(* CODESYS project TcDynCollections.library
   Company: FisoThemes
   DefaultNamespace: TcDynCollections
   Version: 0.2.0.0
   DocFormat: reStructuredText
   Placeholder: TwinCat Dynamic Collections
   Author: Goodwill Mzumala
   Description: A library for handling collections of data dynamically.
   Title: TwinCat Dynamic Collections

Project tree, tasks and I/O mapping:
  libraries: Tc2_Standard, * (Beckhoff Automation GmbH); Tc2_System, * (Beckhoff Automation GmbH); Tc3_Module, * (Beckhoff Automation GmbH); Tc2_Utilities, 3.3.38.0 (Beckhoff Automation GmbH)
  DUTs/
    Interfaces/
      interface I_Collections: _Count, _Error_Status, _Is_Empty, Clear
      interface I_List: Add_Back, Add_Front, Find, Get, Get_First, Get_Value_As_String, Insert, Remove, RemoveAt, Resize, Reverse, Set
      interface I_List_ReadOnly: _Count, _Is_Empty, Find, Get, Get_First, Get_Value_As_String
      interface I_List_WriteOnly: Add_Back, Add_Front, Clear, Insert, Remove, RemoveAt, Resize, Reverse, Set
      interface I_Queue: Dequeue, Dequeue_Void, Enqueue, Enqueue_At_Front, Peek, Reverse
      interface I_Stack: Peek, Pop, Pop_Void, Push, Reverse, Top
    Structs/
      data type ST_ERROR
      data type ST_GENERIC
      data type ST_NODE
  GVLs/
  POUs/
    Examples/
      program P_Array_List_Example [ST]
      program P_List_Example [ST]
      program P_Queue_Example [ST]
      program P_Stack_Example [ST]
    Function Blocks/
      function block FB_Array_List [ST]: ClearException, EmptyListException, LessThanZeroException, MemCmpErrExpection, OutOfBoundsException, TypeMismatchException, CopyValueTo, DecrementCount, Free_Value, GetValueAsString, IncrementCount, Malloc_Array, Malloc_Value, SetValue, _Is_Empty, Add_Back, Add_Front, Clear, FB_exit, FB_init, Find, Get, Get_First, Get_Value_As_String, Insert, Remove, RemoveAt, Resize, Reverse, Set
      function block FB_Collections [ST]: _Count, _Error_Status, _Is_Empty, Clear
      function block FB_List [ST]: ClearException, EmptyListException, MemCmpErrExpection, OutOfBoundsException, TypeMismatchException, CopyValueTo, DecrementCount, Free_Node, GetValueAsString, IncrementCount, Iterate, Malloc_Node, SetValue, _Is_Empty, Add_Back, Add_Front, Clear, FB_exit, FB_init, Find, Get, Get_First, Get_Value_As_String, Insert, Remove, RemoveAt, Resize, Reverse, Set
      function block FB_Queue [ST]: _Count, _Is_Empty, CatchError, Clear, Dequeue, Dequeue_Void, Enqueue, Enqueue_At_Front, Peek, Reverse
      function block FB_Stack [ST]: _Count, _Is_Empty, CatchError, Clear, Peek, Pop, Pop_Void, Push, Reverse, Top
    program MAIN [ST]
  Project Information/
    function F_GetCompany [ST]
    function F_GetTitle [ST]
    function F_GetVersion [ST]
  UML/
    Array List UML
    Collections UML
    List UML
    Queue UML
    Stack UML
  Version/
    global variables Global_Version
  VISUs/
*)

// DUTs/Structs/ST_ERROR
(* STRUCT used to contain error status information. *)
{attribute 'enable_dynamic_creation'}
TYPE ST_ERROR :
STRUCT
	bSTATUS : BOOL; 		// Indicates if an error has occurred | TRUE = error, FALSE = no error
	nCODE 	: DINT; 		// Error code specific to the particular error.
	sSOURCE : T_MaxString; 	// Textual information describing the error.
END_STRUCT
END_TYPE

// DUTs/Structs/ST_GENERIC
(* Generic data type used for Programs/Functions/Function Blocks to handle data in a generic way. *)
{attribute 'enable_dynamic_creation'}
TYPE ST_GENERIC EXTENDS __SYSTEM.AnyType :
STRUCT
	sValue : T_MaxString; 	// Data of parameter as a string for easy convertion.
END_STRUCT
END_TYPE

// DUTs/Structs/ST_NODE
(* Node for linked list*)
{attribute 'enable_dynamic_creation'}
TYPE ST_NODE:
STRUCT
	Data 	: ST_GENERIC; // Stored data.
	pNext 	: POINTER TO ST_NODE := Tc3_Module.GVL.NULL; 	// Pointer to next node.
END_STRUCT
END_TYPE

// Version/Global_Version
{attribute 'TcGenerated'}
{attribute 'no-analysis'}
{attribute 'linkalways'}
// This function has been automatically generated from the project information.
VAR_GLOBAL CONSTANT
	{attribute 'const_non_replaced'}
	stLibVersion_TwinCat_Dynamic_Collections : ST_LibVersion := (iMajor := 0, iMinor := 2, iBuild := 0, iRevision := 0, nFlags := 0, sVersion := '0.2.0.0');
END_VAR

// DUTs/Interfaces/I_Collections
INTERFACE I_Collections

// Number of items in the collection
PROPERTY _Count : DINT
GET
END_GET
END_PROPERTY

(* Gets collection's error status *)
PROPERTY _Error_Status : ST_ERROR
GET
END_GET
END_PROPERTY

// Checks if collection is empty
PROPERTY _Is_Empty : BOOL
GET
END_GET
END_PROPERTY

// Empties/Clears/Deletes every item in the collection
METHOD Clear
END_METHOD

END_INTERFACE

// DUTs/Interfaces/I_List
INTERFACE I_List EXTENDS I_Collections

// Adds an item to the end of the list
METHOD Add_Back : I_List
VAR_INPUT
	Item 	: ANY; // Item to store in list
END_VAR
END_METHOD

// Adds an item at the front of the list
METHOD Add_Front : I_List
VAR_INPUT
	Item 	: ANY; // Item to store in list
END_VAR
END_METHOD

// Find the location of an item in list.
METHOD Find : I_List
VAR_INPUT
	Item 	: ANY; // Item to find in list
END_VAR
VAR_OUTPUT
	nIndex	: DINT; //Location of item in list 
END_VAR
END_METHOD

// Gets item from list at specified location without removing it
METHOD Get : I_List
VAR_INPUT
	Return_Item 	: ANY;  // Variable to store returned item
	nIndex 			: DINT; // Location of item
END_VAR
END_METHOD

// Gets item at the front of the list 
METHOD Get_First : I_List
VAR_INPUT
	Return_Item 	: ANY; // Variable to store returned item
END_VAR
END_METHOD

// Returns item as a string, if type to string conversion is supported
METHOD Get_Value_As_String : I_List
VAR_INPUT
	nIndex	: DINT; // Location of item
END_VAR
VAR_OUTPUT
	sItem 	: T_MaxString; // Variable to store returned item
END_VAR
END_METHOD

// Adds new item to list at specified location, if index = 0, item will be added at the front, if index = count, item will be added at the back
METHOD Insert : I_List
VAR_INPUT
	Item 	: ANY;  // Item to store in list
	nIndex 	: DINT; // Location of item
END_VAR
END_METHOD

// Removes item at the front of the list and returns nothing
METHOD Remove : I_List
END_METHOD

// Remove item at specified location and return nothing
METHOD RemoveAt : I_List
VAR_INPUT
	nIndex : DINT; // Location of item
END_VAR
END_METHOD

// Manually resize list. If list becomes smaller, items on higher locations will be deleted.
METHOD Resize : I_List
VAR_INPUT
	nSize : DINT; // New size of list.
END_VAR
END_METHOD

// Reverses the order of items in the list
METHOD Reverse : I_List
END_METHOD

// Adds new item to list in the specified location without resizing list
METHOD Set : I_List
VAR_INPUT
	Item 	: ANY; 	// Item to store in list
	nIndex 	: DINT; // Location of item
END_VAR
END_METHOD

END_INTERFACE

// DUTs/Interfaces/I_List_ReadOnly
// Implement this with I_List to allow a list to be Read Only. 
INTERFACE I_List_ReadOnly

// Number of items in the collection
PROPERTY _Count : DINT
GET
END_GET
END_PROPERTY

// Checks if collection is empty
PROPERTY _Is_Empty : BOOL
GET
END_GET
END_PROPERTY

// Find the location of an item in list.
METHOD Find : I_List
VAR_INPUT
	Item 	: ANY; // Item to find in list
END_VAR
VAR_OUTPUT
	nIndex	: DINT; //Location of item in list 
END_VAR
END_METHOD

// Gets item from list at specified location without removing it
METHOD Get : I_List
VAR_INPUT
	Return_Item 	: ANY;  // Variable to store returned item
	nIndex 			: DINT; // Location of item
END_VAR
END_METHOD

// Gets item at the front of the list 
METHOD Get_First : I_List
VAR_INPUT
	Return_Item 	: ANY; // Variable to store returned item
END_VAR
END_METHOD

// Returns item as a string, if type to string conversion is supported
METHOD Get_Value_As_String : I_List
VAR_INPUT
	nIndex	: DINT; // Location of item
END_VAR
VAR_OUTPUT
	sItem 	: T_MaxString; // Variable to store returned item
END_VAR
END_METHOD

END_INTERFACE

// DUTs/Interfaces/I_List_WriteOnly
// Implement this with I_List to allow a list to be Write Only. 
INTERFACE I_List_WriteOnly

// Adds an item to the end of the list
METHOD Add_Back : I_List
VAR_INPUT
	Item 	: ANY; // Item to store in list
END_VAR
END_METHOD

// Adds an item at the front of the list
METHOD Add_Front : I_List
VAR_INPUT
	Item 	: ANY; // Item to store in list
END_VAR
END_METHOD

// Empties/Clears/Deletes every item in the collection
METHOD Clear
END_METHOD

// Adds new item to list at specified location, if index = 0, item will be added at the front, if index = count, item will be added at the back
METHOD Insert : I_List
VAR_INPUT
	Item 	: ANY;  // Item to store in list
	nIndex 	: DINT; // Location of item
END_VAR
END_METHOD

// Removes item at the front of the list and returns nothing
METHOD Remove : I_List
END_METHOD

// Remove item at specified location and return nothing
METHOD RemoveAt : I_List
VAR_INPUT
	nIndex : DINT; // Location of item
END_VAR
END_METHOD

// Manually resize list. If list becomes smaller, items on higher locations will be deleted.
METHOD Resize : I_List
VAR_INPUT
	nSize : DINT; // New size of list.
END_VAR
END_METHOD

// Reverses the order of items in the list
METHOD Reverse : I_List
END_METHOD

// Adds new item to list in the specified location without resizing list
METHOD Set : I_List
VAR_INPUT
	Item 	: ANY; 	// Item to store in list
	nIndex 	: DINT; // Location of item
END_VAR
END_METHOD

END_INTERFACE

// DUTs/Interfaces/I_Queue
INTERFACE I_Queue EXTENDS I_Collections

(* Gets and remove item at the front of the queue *)
METHOD Dequeue : I_Queue
VAR_INPUT
	Item : ANY; (* Variable to store returned item value *)
END_VAR
END_METHOD

(* Removes item at the front of the queue without returning anything *)
METHOD Dequeue_Void : I_Queue
VAR_INPUT
END_VAR
END_METHOD

(* Adds item at the back of the queue *)
METHOD Enqueue : I_Queue
VAR_INPUT
	Item : ANY; (* Variable containg data to store on the queue *)
END_VAR
END_METHOD

(* Adds item at the front of the queue *)
METHOD Enqueue_At_Front : I_Queue
VAR_INPUT
	Item : ANY; (* Variable containg data to store on the queue *)
END_VAR
END_METHOD

(* Get item from the queue without removing it. *)
METHOD Peek : I_Queue
VAR_INPUT
	Item 	: ANY; (* Variable to store returned item value *)
	nIndex 	: DINT; (* Location of item*)
END_VAR
END_METHOD

METHOD Reverse : I_Queue
VAR_INPUT
END_VAR
END_METHOD

END_INTERFACE

// DUTs/Interfaces/I_Stack
INTERFACE I_Stack EXTENDS I_Collections

(* Get item from stack without removing it. *)
METHOD Peek : I_Stack
VAR_INPUT
	Item 	: ANY; (* Variable to store returned item value *)
	nIndex 	: DINT; (* Location of item*)
END_VAR
END_METHOD

(* Gets and deletes item at the top of the stack *)
METHOD Pop : I_Stack
VAR_INPUT
	Item : ANY; (* Variable to store returned item value *)
END_VAR
END_METHOD

(* Removes item at the top of the stack without returning anything *)
METHOD Pop_Void : I_Stack
VAR_INPUT
END_VAR
END_METHOD

(* Add item to the top of the stack *)
METHOD Push : I_Stack
VAR_INPUT
	Item : ANY; (* Variable containg data to store on the stack *)
END_VAR
END_METHOD

(* Reverses order of items on stack *)
METHOD Reverse : I_Stack
VAR_INPUT
END_VAR
END_METHOD

(* Get item at the top of the stack without removing it. *)
METHOD Top : I_Stack
VAR_INPUT
	Item 	: ANY; (* Variable to store returned item value *)
END_VAR
END_METHOD

END_INTERFACE

// POUs/Examples/P_Array_List_Example
PROGRAM P_Array_List_Example
VAR
	eState 		: (IDLE, INSERT, REVERSE, RESIZE, GET, SET, FIND, CLEAR, ADD_FRONT, ADD_BACK, REMOVE, REMOVE_AT);
	fbArray_List: FB_Array_List(0);
	nFind 		: DINT;
	sData 		: WSTRING;
	sRTNData	: ARRAY[0..6] OF WSTRING;
	nCount 		: DINT;
	stError 	: ST_ERROR;
END_VAR

stError := fbArray_List._Error_Status;
CASE eState OF
	INSERT:
		sData := "Cats";	fbArray_List.Insert(sData, 0);
		sData := "Dogs";	fbArray_List.Insert(sData, 1);
		sData := "Ravens";	fbArray_List.Insert(sData, 2);
		sData := "Mollies";	fbArray_List.Insert(sData, 3);
	REVERSE:
		fbArray_List.Reverse();
	RESIZE:
		fbArray_List.Resize(3);
	GET: 
		fbArray_List
			.Get(sRTNData[0], 0)
			.Get(sRTNData[1], 1)
			.Get(sRTNData[2], 2)
			.Get(sRTNData[3], 3)
			.Get(sRTNData[4], 4)
			.Get(sRTNData[5], 5)
			.Get(sRTNData[6], 6);
	SET:
		sData := "Ravens";	fbArray_List.Set(sData, 0);
		sData := "Mollies";	fbArray_List.Set(sData, 1);
		sData := "Dogs";	fbArray_List.Set(sData, 2);
		sData := "Cats";	fbArray_List.Set(sData, 3);
	FIND:
		sData := "Dogs"; fbArray_List.Find(sData, nIndex => nFind);
	CLEAR:
		fbArray_List.Clear();
	ADD_FRONT:
		sData := "Pythons";fbArray_List.Add_Front(sData);
	ADD_BACK:
		sData := "Anacondas"; fbArray_List.Add_Back(sData);
	REMOVE:
		fbArray_List.Remove();
	REMOVE_AT:
		fbArray_List.RemoveAt(2);
END_CASE
nCount := fbArray_List._Count;
eState := IDLE;

END_PROGRAM

// POUs/Function Blocks/FB_Array_List
(* A dynamic array that holds data of multiple types and can grow or shrink at run time. *)
FUNCTION_BLOCK FB_Array_List EXTENDS FB_Collections IMPLEMENTS I_List, I_List_ReadOnly, I_List_WriteOnly
VAR
	pData 		: POINTER TO ST_GENERIC;
END_VAR
VAR CONSTANT
	{warning disable C0228}
	stData 		: ST_GENERIC := (TypeClass := __SYSTEM.TYPE_CLASS.TYPE_NONE);
END_VAR

METHOD PROTECTED ClearException : BOOL;
VAR
END_VAR
ClearException 	:= stError.bSTATUS := FALSE;
stError.nCODE 	:= 0;
stError.sSOURCE := 'No error.';
END_METHOD

// Raises an expection if list is empty
METHOD PROTECTED EmptyListException : BOOL
VAR_INPUT
END_VAR
IF THIS^._Is_Empty THEN
	stError.bSTATUS := TRUE;
	stError.nCODE 	:= 2936;
	stError.sSOURCE := 'List is empty';
ELSE
	This^.ClearException();
	END_IF
EmptyListException := stError.bSTATUS;
END_METHOD

METHOD PROTECTED LessThanZeroException : BOOL
VAR_INPUT
	nIndex : DINT;
END_VAR
IF (nIndex < 0) THEN
	stError.bSTATUS := TRUE;
	stError.nCODE 	:= 5365;
	stError.sSOURCE := 'Out of bounds. Index is less than zero.';
ELSE
	This^.ClearException();
	END_IF
LessThanZeroException := stError.bSTATUS;
END_METHOD

// Compares memory sizes of 2 addresses. Returns TRUE  and raises error flag if theyre not same size.
METHOD PROTECTED MemCmpErrExpection : BOOL
VAR_INPUT
	pDestAddr,
	pSrcAddr 	: PVOID;
	nSize 		: UDINT;
END_VAR
VAR_INST
	nMemErr : DINT;
END_VAR
nMemErr := MEMCMP(pDestAddr, pSrcAddr, nSize);
IF nMemErr = -1 THEN 
	stError.bSTATUS := TRUE;
	stError.nCODE 	:= 4129;
	stError.sSOURCE := 'Incorrect parameter values. Destination address smaller than source address';
	
ELSIF nMemErr = 0 THEN THIS^.ClearException();
	
ELSIF nMemErr = 1 THEN
	stError.bSTATUS := TRUE;
	stError.nCODE 	:= 4823;
	stError.sSOURCE := 'Incorrect parameter values. Destination address greater that source address';

ELSE
	stError.bSTATUS := TRUE;
	stError.nCODE 	:= 4564;
	stError.sSOURCE := 'Incorrect parameter values. Pointer to destination/source address is NULL or allocated address memory is NULL.';
	END_IF

MemCmpErrExpection := stError.bSTATUS;
END_METHOD

METHOD PROTECTED OutOfBoundsException : BOOL
VAR_INPUT
	nIndex : DINT;
END_VAR
IF (nIndex < 0) OR (nIndex >= THIS^._Count) THEN
	stError.bSTATUS := TRUE;
	stError.nCODE 	:= 5374;
	stError.sSOURCE := 'Out of bounds. You tried to access data outside the range of this list.';
ELSE
	This^.ClearException();
	END_IF
OutOfBoundsException := stError.bSTATUS;
END_METHOD

METHOD TypeMismatchException : BOOL
VAR_INPUT
	Dest,
	Src 	: __SYSTEM.AnyType;
END_VAR
IF Dest.diSize <> Src.diSize THEN
	stError.bSTATUS := TRUE;
	stError.nCODE 	:= 3172;
	stError.sSOURCE := 'Type mismatch. Byte sizes are not the same';
ELSIF Dest.TypeClass <> Src.TypeClass THEN
	stError.bSTATUS := TRUE;
	stError.nCODE 	:= 3172;
	stError.sSOURCE := 'Type mismatch. Type classes are not the same';
ELSE
	THIS^.ClearException();
END_IF
TypeMismatchException := stError.bSTATUS;
END_METHOD

// Copy data from source memory space to desination memory space
METHOD PROTECTED CopyValueTo
VAR_INPUT
	Dest, Src 	: __SYSTEM.AnyType;
END_VAR
MEMMOVE(Dest.pValue, Src.pValue, TO_UDINT(Src.diSize));
END_METHOD

// Decrement list size by 1.
METHOD PROTECTED DecrementCount
VAR_INPUT
END_VAR
THIS^.nCount := THIS^.nCount - 1;
END_METHOD

// Deletes/frees Generic value's value from memory
METHOD PROTECTED Free_Value
VAR_INPUT
	Variable : __SYSTEM.AnyType;
END_VAR
IF Variable.pValue = 0 THEN RETURN; END_IF
__DELETE(Variable.pValue);
END_METHOD

METHOD PROTECTED GetValueAsString : T_MaxString
VAR_INPUT
	 Value : __SYSTEM.AnyType;
END_VAR
VAR	
	pBool			: POINTER TO BOOL;
    pByte			: POINTER TO BYTE;
    pWord			: POINTER TO WORD;
    pDWord			: POINTER TO DWORD;
    pLWord			: POINTER TO LWORD;
    pSint			: POINTER TO SINT;
    pInt			: POINTER TO INT;
    pDint			: POINTER TO DINT;
    pLint			: POINTER TO LINT;
    pUSint			: POINTER TO USINT;
    pUInt			: POINTER TO UINT;
    pUDint			: POINTER TO UDINT;
    pULint			: POINTER TO ULINT;
    pReal			: POINTER TO REAL;
    pLReal			: POINTER TO LREAL;
    pString			: POINTER TO STRING(255);
    pWString		: POINTER TO WSTRING;
    pTime			: POINTER TO TIME;
    pDate			: POINTER TO DATE;
    pDate_And_Time	: POINTER TO DATE_AND_TIME;
    pTime_Of_Day	: POINTER TO TIME_OF_DAY;
    pPointer		: PVOID;
	pLTime 			: POINTER TO LTIME;
END_VAR
IF Value.pValue = 0 THEN GetValueAsString := 'NULL'; RETURN; END_IF;

CASE Value.TypeClass OF 
	__SYSTEM.TYPE_CLASS.TYPE_BOOL:
		pBool := Value.pValue;
		GetValueAsString := TO_STRING(pBool^);
		
    __SYSTEM.TYPE_CLASS.TYPE_BYTE:
		pByte := Value.pValue;
		GetValueAsString := TO_STRING(pByte^);
		
    __SYSTEM.TYPE_CLASS.TYPE_WORD:
		pWord := Value.pValue;
		GetValueAsString := TO_STRING(pWord^);
		
    __SYSTEM.TYPE_CLASS.TYPE_DWORD:
		pDWord := Value.pValue;
		GetValueAsString := TO_STRING(pDWord^);
		
    __SYSTEM.TYPE_CLASS.TYPE_LWORD:
		pLWord := Value.pValue;
		GetValueAsString := TO_STRING(pLWord^);
		
    __SYSTEM.TYPE_CLASS.TYPE_SINT:
		pSint := Value.pValue;
		GetValueAsString := TO_STRING(pSint^);
		
    __SYSTEM.TYPE_CLASS.TYPE_INT:
		pInt := Value.pValue;
		GetValueAsString := TO_STRING(pInt^);
		
    __SYSTEM.TYPE_CLASS.TYPE_DINT:
		pDint := Value.pValue;
		GetValueAsString := TO_STRING(pDint^);
		
    __SYSTEM.TYPE_CLASS.TYPE_LINT:
		pLint := Value.pValue;
		GetValueAsString := TO_STRING(pLint^);
		
    __SYSTEM.TYPE_CLASS.TYPE_USINT:
		pUSint := Value.pValue;
		GetValueAsString := TO_STRING(pUSint^);
		
    __SYSTEM.TYPE_CLASS.TYPE_UINT:
		pUInt := Value.pValue;
		GetValueAsString := TO_STRING(pUInt^);
		
    __SYSTEM.TYPE_CLASS.TYPE_UDINT:
		pUDint := Value.pValue;
		GetValueAsString := TO_STRING(pUDint^);
		
    __SYSTEM.TYPE_CLASS.TYPE_ULINT:
		pULint := Value.pValue;
		GetValueAsString := TO_STRING(pULint^);
		
   __SYSTEM.TYPE_CLASS.TYPE_REAL:
		pReal := Value.pValue;
		GetValueAsString := TO_STRING(pReal^);
		
    __SYSTEM.TYPE_CLASS.TYPE_LREAL:
		pLReal := Value.pValue;
		GetValueAsString := TO_STRING(pLReal^);
		
    __SYSTEM.TYPE_CLASS.TYPE_STRING:
		pString := Value.pValue;
		GetValueAsString := TO_STRING(pString^);
		
   __SYSTEM.TYPE_CLASS.TYPE_WSTRING:
		pWString := Value.pValue;
		GetValueAsString := TO_STRING(pWString^);
		
    __SYSTEM.TYPE_CLASS.TYPE_TIME:
		pTime := Value.pValue;
		GetValueAsString := TO_STRING(pTime^);
		
    __SYSTEM.TYPE_CLASS.TYPE_DATE:
		pDate := Value.pValue;
		GetValueAsString := TO_STRING(pDate^);
		
    __SYSTEM.TYPE_CLASS.TYPE_DATEANDTIME:
		pDate_And_Time := Value.pValue;
		GetValueAsString := TO_STRING(pDate_And_Time^);
		
    __SYSTEM.TYPE_CLASS.TYPE_TIMEOFDAY:
		pTime_Of_Day := Value.pValue;
		GetValueAsString := TO_STRING(pTime_Of_Day^);
	
	__SYSTEM.TYPE_CLASS.TYPE_POINTER:
		GetValueAsString := TO_STRING(Value.pValue);
		
	__SYSTEM.TYPE_CLASS.TYPE_LTIME:
		pLTime := Value.pValue;
		GetValueAsString := TO_STRING(pLTime^);
ELSE
	GetValueAsString := 'TYPE TO STRING CONVERSION NOT SUPPORTED BY THIS TYPE'; 
END_CASE
END_METHOD

// Increments list size by 1
METHOD PROTECTED IncrementCount
VAR_INPUT
END_VAR
THIS^.nCount := THIS^.nCount + 1;
END_METHOD

// Allocate memory space for Array of Generics on the heap, returns Pointer to start of Generic Array;
// WARNING!!! Always have a place to store the return otherwise a memory leak will occur.
METHOD PROTECTED Malloc_Array : POINTER TO ST_GENERIC
VAR_INPUT
	nSize : DINT; // Array Size
END_VAR
VAR
	i, nByte_Size: DINT;
END_VAR
VAR CONSTANT
	{warning disable C0228}
	stData 		: ST_GENERIC;
END_VAR
nByte_Size := SIZEOF(ST_GENERIC)*nSize;
Malloc_Array := __NEW(BYTE, TO_UDINT(nByte_Size));
END_METHOD

// Allocate memory space for the Generic value's data on the heap, returns Generic;
// WARNING!!! Always have a place to store the return otherwise a memory leak will occur.
METHOD PROTECTED Malloc_Value : ST_GENERIC
VAR_INPUT
	Variable : __SYSTEM.AnyType;
END_VAR
Malloc_Value.sValue 	:= THIS^.GetValueAsString(Variable);
Malloc_Value.pValue 	:= __NEW(BYTE, TO_UDINT(Variable.diSize)); // Allocate space in memory to store data value.
Malloc_Value.diSize 	:= Variable.diSize;
Malloc_Value.TypeClass 	:= Variable.TypeClass;
END_METHOD

(* Set value of __SYSTEM.Anytype variable *)
METHOD PROTECTED SetValue
VAR_INPUT
	Variable	: __SYSTEM.Anytype;
	Value 		: USINT; // Character/byte to set.
END_VAR
MEMSET(Variable.pValue, Value, TO_UDINT(Variable.diSize));
END_METHOD

(* Checks of list is empty.*)
PROPERTY _Is_Empty : BOOL
GET
_Is_Empty := THIS^.nCount = 0;
END_GET
END_PROPERTY

// Adds an item to the end of the list
METHOD Add_Back : I_List
VAR_INPUT
	Item 	: ANY; // Item to store in list
END_VAR
Add_Back := THIS^;
IF THIS^._Is_Empty THEN THIS^.FB_init(FALSE,FALSE, 1); THIS^.Set(Item, 0); RETURN; END_IF
THIS^.Resize(THIS^._Count+1);
THIS^.Free_Value(THIS^.pData[THIS^._Count-1]);
THIS^.pData[THIS^._Count-1] := THIS^.Malloc_Value(Item);
THIS^.CopyValueTo(THIS^.pData[THIS^._Count-1], Item);
END_METHOD

// Adds an item at the front of the list
METHOD Add_Front : I_List
VAR_INPUT
	Item 	: ANY; // Item to store in list
END_VAR
VAR
	pOld_Data : POINTER TO ST_GENERIC;
	i : DINT;
END_VAR
Add_Front := THIS^;
IF THIS^._Is_Empty THEN THIS^.FB_init(FALSE,FALSE, 1); THIS^.Set(Item, 0); RETURN; END_IF

pOld_Data := THIS^.pData;
THIS^.pData := THIS^.Malloc_Array(THIS^._Count+1);

FOR i := 1 TO THIS^._Count DO
	THIS^.pData[i] := THIS^.Malloc_Value(pOld_Data[i-1]);
	THIS^.CopyValueTo(THIS^.pData[i], pOld_Data[i-1]);
	THIS^.Free_Value(pOld_Data[i-1]);
	END_FOR
__DELETE(pOld_Data);
THIS^.Set(Item, 0);
THIS^.IncrementCount();
END_METHOD

// Empties/Clears/Deletes every item in the list
METHOD Clear
VAR
	i : DINT;
END_VAR
IF NOT(THIS^._Is_Empty) THEN 
	FOR i := 0 TO THIS^._Count - 1 DO THIS^.Free_Value(THIS^.pData[i]); END_FOR
	__DELETE(THIS^.pData); 
	THIS^.nCount := 0; 
	END_IF
END_METHOD

METHOD FB_exit : BOOL
VAR_INPUT
	bInCopyCode : BOOL; // if TRUE, the exit method is called for exiting an instance that is copied afterwards (online change).
END_VAR
THIS^.Clear();
END_METHOD

METHOD FB_init : BOOL
VAR_INPUT
	bInitRetains 	: BOOL; // if TRUE, the retain variables are initialized (warm start / cold start)
	bInCopyCode 	: BOOL; // if TRUE, the instance afterwards gets moved into the copy code (online change)
	nLength 		: DINT; // Length to initialise array with.
END_VAR
VAR
	i, nByte_Size 	: DINT;
END_VAR
THIS^.Clear();
IF nLength <= 0 THEN RETURN; END_IF
THIS^.nCount := nLength;
THIS^.pData := THIS^.Malloc_Array(nLength);
END_METHOD

// Find the location of an item in list.
METHOD Find : I_List
VAR_INPUT
	Item 	: ANY; // Item to find in list
END_VAR
VAR_OUTPUT
	nIndex	: DINT; //Location of item in list 
END_VAR
VAR
	i : DINT;
	n : DINT := -1;
END_VAR
Find := THIS^;
IF THIS^.EmptyListException() THEN nIndex := -1; RETURN; END_IF
FOR i := 0 TO THIS^._Count-1 DO
	IF (THIS^.pData[i].pValue = 0) 					 THEN CONTINUE; END_IF
	IF (Item.TypeClass <> THIS^.pData[i].TypeClass) THEN CONTINUE; END_IF
	IF (Item.pValue^ <> THIS^.pData[i].pValue^) 	 THEN CONTINUE; END_IF
	
	CASE Item.TypeClass OF
		__SYSTEM.TYPE_CLASS.TYPE_STRING:
			IF LEN2(Item.pValue) <> LEN2(THIS^.pData[i].pValue) THEN CONTINUE; END_IF
			n := MEMCMP(Item.pValue, THIS^.pData[i].pValue, LEN2(THIS^.pData[i].pValue)+1);
				
		__SYSTEM.TYPE_CLASS.TYPE_WSTRING:
			IF WLEN2(Item.pValue) <> WLEN2(THIS^.pData[i].pValue) THEN CONTINUE; END_IF
			n := MEMCMP(Item.pValue, THIS^.pData[i].pValue, (WLEN2(THIS^.pData[i].pValue)*SIZEOF(WORD))+1);
	ELSE
		IF (Item.diSize <> THIS^.pData[i].diSize) THEN CONTINUE; END_IF	
		n := MEMCMP(Item.pValue, THIS^.pData[i].pValue, TO_UDINT(Item.diSize));
		END_CASE
		IF n = 0 THEN nIndex := i; RETURN; END_IF
	END_FOR
nIndex := -1;
END_METHOD

// Gets item at specified location;
METHOD Get : I_List
VAR_INPUT
	Return_Item 	: ANY;  // Variable to store requested node value
	nIndex 			: DINT; // Location of node
END_VAR
VAR_INST
	data : ST_GENERIC;
END_VAR
Get := THIS^;
IF THIS^.EmptyListException() OR THIS^.OutOfBoundsException(nIndex) THEN THIS^.SetValue(Return_Item, 16#0); RETURN; END_IF
IF THIS^.TypeMismatchException(Return_Item, THIS^.pData[nIndex]) THEN THIS^.SetValue(Return_Item, 16#0); RETURN; END_IF
THIS^.CopyValueTo(Return_Item, THIS^.pData[nIndex]);
END_METHOD

// Gets item at the front of the list 
METHOD Get_First : I_List
VAR_INPUT
	Return_Item 	: ANY; // Variable to store returned item
END_VAR
Get_First := THIS^;
THIS^.Get(Return_Item, 0);
END_METHOD

// Returns item as a string, if type to string conversion is supported
METHOD Get_Value_As_String : I_List
VAR_INPUT
	nIndex	: DINT; // Location of item
END_VAR
VAR_OUTPUT
	sItem 	: T_MaxString; // Variable to store returned item
END_VAR
Get_Value_As_String := THIS^;
IF THIS^.EmptyListException() OR THIS^.OutOfBoundsException(nIndex) THEN sItem := 'ERR: List is Empty or index Out of Bounds'; RETURN; END_IF
sItem := THIS^.pData[nIndex].sValue;
END_METHOD

// Adds new item to list at specified location, if index = 0, item will be added at the front, if index = count, item will be added at the back
METHOD Insert : I_List
VAR_INPUT
	Item 	: ANY;  // Item to store in list
	nIndex 	: DINT; // Location of item
END_VAR
VAR
	pOld_Data : POINTER TO ST_GENERIC;
	i : DINT;
END_VAR
Insert := THIS^;
IF nIndex = 0 THEN THIS^.Add_Front(Item); RETURN; END_IF
IF nIndex = THIS^._Count THEN THIS^.Add_Back(Item); RETURN; END_IF
IF THIS^.OutOfBoundsException(nIndex) THEN RETURN; END_IF

pOld_Data := THIS^.pData;
THIS^.pData := THIS^.Malloc_Array(THIS^._Count+1);
THIS^.IncrementCount();

FOR i := 0 TO nIndex-1 DO
	THIS^.pData[i] := THIS^.Malloc_Value(pOld_Data[i]);
	THIS^.CopyValueTo(THIS^.pData[i], pOld_Data[i]);
	THIS^.Free_Value(pOld_Data[i]);
	END_FOR
	
THIS^.Set(Item, nIndex);
	
FOR i := nIndex+1 TO THIS^._Count-1 DO
	THIS^.pData[i] := THIS^.Malloc_Value(pOld_Data[i-1]);
	THIS^.CopyValueTo(THIS^.pData[i], pOld_Data[i-1]);
	THIS^.Free_Value(pOld_Data[i-1]);
	END_FOR
__DELETE(pOld_Data);
END_METHOD

// Removes item at the front of the list and returns nothing
METHOD Remove : I_List
VAR
	i : DINT;
END_VAR
Remove := THIS^;
IF THIS^.EmptyListException() THEN RETURN; END_IF
IF THIS^._Count = 1 THEN THIS^.Clear(); RETURN; END_IF;
THIS^.Free_Value(THIS^.pData[0]);
FOR i := 0 TO THIS^._Count-2 DO THIS^.pData[i] := THIS^.pData[i+1]; END_FOR
THIS^.Resize(THIS^._Count-1);
END_METHOD

// Remove item at specified location and return nothing
METHOD RemoveAt : I_List
VAR_INPUT
	nIndex : DINT; // Location of item
END_VAR
VAR
	i : DINT;
END_VAR
RemoveAt := THIS^;
IF THIS^.EmptyListException() THEN RETURN; END_IF
IF THIS^.OutOfBoundsException(nIndex) THEN RETURN; END_IF
IF nIndex = 0 THEN THIS^.Remove(); RETURN; END_IF
IF nIndex = THIS^._Count - 1 THEN THIS^.Resize(THIS^._Count - 1); RETURN; END_IF
THIS^.Free_Value(THIS^.pData[nIndex]);
FOR i := nIndex TO THIS^._Count-1 DO THIS^.pData[i] := THIS^.pData[i+1]; END_FOR
THIS^.Resize(THIS^._Count-1);
END_METHOD

// Manually resize list. If list becomes smaller, items on higher locations will be deleted.
METHOD Resize : I_List
VAR_INPUT
	nSize : DINT; // New size of list.
END_VAR
VAR
	pOld_Data 		: POINTER TO ST_GENERIC;
	i,
	nOld_Data_Count, 
	nByte_Size : DINT;
END_VAR
Resize := THIS^;
IF THIS^.LessThanZeroException(nSize) THEN RETURN; END_IF
IF (nSize = 0) THEN THIS^.Clear(); RETURN; END_IF
IF nSize = THIS^._Count THEN RETURN; END_IF
IF THIS^._Is_Empty THEN THIS^.FB_init(FALSE,FALSE, nSize); RETURN; END_IF

pOld_Data 		:= THIS^.pData;
nOld_Data_Count := THIS^._Count;

THIS^.pData := THIS^.Malloc_Array(nSize);

FOR i := 0 TO nSize - 1 DO
	IF (i = nOld_Data_Count) AND (nSize > nOld_Data_Count) THEN EXIT; END_IF
	THIS^.pData[i] := THIS^.Malloc_Value(pOld_Data[i]);
	THIS^.CopyValueTo(THIS^.pData[i], pOld_Data[i]);
	THIS^.Free_Value(pOld_Data[i]);
	END_FOR
__DELETE(pOld_Data);
THIS^.nCount := nSize;
END_METHOD

// Reverses the order of items in the list
METHOD Reverse : I_List
VAR
	pOld_Data 	: POINTER TO ST_GENERIC;
	nByte_Size 	: DINT;
	i			: DINT;
END_VAR
Reverse := THIS^;
IF THIS^.EmptyListException() THEN RETURN; END_IF
IF THIS^._Count = 1 THEN RETURN; END_IF

pOld_Data 	:= THIS^.pData;

THIS^.pData := THIS^.Malloc_Array(THIS^._Count);

FOR i:= 0 TO THIS^._Count - 1 DO
	THIS^.pData[i] := THIS^.Malloc_Value(pOld_Data[(THIS^._Count-1)-i]);
	THIS^.CopyValueTo(THIS^.pData[i], pOld_Data[(THIS^._Count-1)-i]);
	THIS^.Free_Value(pOld_Data[(THIS^._Count-1)-i]);
	END_FOR
__DELETE(pOld_Data);
END_METHOD

// Adds new item to list in the specified location without resizing list
METHOD Set : I_List
VAR_INPUT
	Item 	: ANY; 	// Item to store in list
	nIndex 	: DINT; // Location of item
END_VAR
Set := THIS^;
IF THIS^.OutOfBoundsException(nIndex) OR THIS^.EmptyListException() THEN RETURN; END_IF
THIS^.Free_Value(THIS^.pData[nIndex]);
THIS^.pData[nIndex] := THIS^.Malloc_Value(Item);
THIS^.CopyValueTo(THIS^.pData[nIndex], Item);
END_METHOD

END_FUNCTION_BLOCK

// POUs/Function Blocks/FB_Collections
FUNCTION_BLOCK ABSTRACT FB_Collections IMPLEMENTS I_Collections
VAR
	stError : ST_ERROR;
	nCount 	: DINT; // Size of Collection
END_VAR

(* Number of items in the collection *)
PROPERTY _Count : DINT
GET
_Count := THIS^.nCount;
END_GET
END_PROPERTY

(* Gets collection's error status *)
PROPERTY _Error_Status : ST_ERROR
GET
_Error_Status := THIS^.stError;
END_GET
END_PROPERTY

(* Checks if collection is empty.*)
PROPERTY _Is_Empty : BOOL
GET
END_GET
END_PROPERTY

(* Empties/Clears/Deletes every element on the collection*)
METHOD Clear
END_METHOD

END_FUNCTION_BLOCK

// POUs/Examples/P_List_Example
PROGRAM P_List_Example
VAR
	eState 		: (IDLE, INSERT, REVERSE, RESIZE, GET, SET, FIND, CLEAR, ADD_FRONT, ADD_BACK, REMOVE, REMOVE_AT);
	fbList 		: FB_List;
	nFind 		: DINT;
	sData 		: WSTRING;
	sRTNData	: ARRAY[0..6] OF WSTRING;
	nCount 		: DINT;
	stError 	: ST_ERROR;
END_VAR

stError := fbList._Error_Status;
CASE eState OF
	INSERT:
		sData := "Cats";	fbList.Insert(sData, 0);
		sData := "Dogs";	fbList.Insert(sData, 1);
		sData := "Ravens";	fbList.Insert(sData, 2);
		sData := "Mollies";	fbList.Insert(sData, 3);
	REVERSE:
		fbList.Reverse();
	RESIZE:
		fbList.Resize(3);
	GET: 
		fbList
			.Get(sRTNData[0], 0)
			.Get(sRTNData[1], 1)
			.Get(sRTNData[2], 2)
			.Get(sRTNData[3], 3)
			.Get(sRTNData[4], 4)
			.Get(sRTNData[5], 5)
			.Get(sRTNData[6], 6);
	SET:
		sData := "Ravens";	fbList.Set(sData, 0);
		sData := "Mollies";	fbList.Set(sData, 1);
		sData := "Dogs";	fbList.Set(sData, 2);
		sData := "Cats";	fbList.Set(sData, 3);
	FIND:
		sData := "Dogs"; fbList.Find(sData, nIndex => nFind);
	CLEAR:
		fbList.Clear();
	ADD_FRONT:
		sData := "Pythons";fbList.Add_Front(sData);
	ADD_BACK:
		sData := "Anacondas"; fbList.Add_Back(sData);
	REMOVE:
		fbList.Remove();
	REMOVE_AT:
		fbList.RemoveAt(2);
END_CASE
nCount := fbList._Count;
eState := IDLE;

END_PROGRAM

// POUs/Function Blocks/FB_List
// Dyanamic List that can store a collection of any types. Similiar to python lists.
FUNCTION_BLOCK FB_List EXTENDS FB_Collections IMPLEMENTS I_List, I_List_ReadOnly, I_List_WriteOnly
VAR
	pHead	: POINTER TO ST_NODE;
END_VAR

METHOD PROTECTED ClearException : BOOL;
VAR
END_VAR
ClearException 	:= stError.bSTATUS := FALSE;
stError.nCODE 	:= 0;
stError.sSOURCE := 'No error.';
END_METHOD

// Raises an expection if list is empty
METHOD PROTECTED EmptyListException : BOOL
VAR_INPUT
END_VAR
IF THIS^._Is_Empty THEN
	stError.bSTATUS := TRUE;
	stError.nCODE 	:= 2936;
	stError.sSOURCE := 'List is empty';
ELSE
	This^.ClearException();
	END_IF
EmptyListException := stError.bSTATUS;
END_METHOD

// Compares memory sizes of 2 addresses. Returns TRUE  and raises error flag if theyre not same size.
METHOD PROTECTED MemCmpErrExpection : BOOL
VAR_INPUT
	pDestAddr,
	pSrcAddr 	: PVOID;
	nSize 		: UDINT;
END_VAR
VAR_INST
	nMemErr : DINT;
END_VAR
nMemErr := MEMCMP(pDestAddr, pSrcAddr, nSize);
IF nMemErr = -1 THEN 
	stError.bSTATUS := TRUE;
	stError.nCODE 	:= 4129;
	stError.sSOURCE := 'Incorrect parameter values. Destination address smaller than source address';
	
ELSIF nMemErr = 0 THEN THIS^.ClearException();
	
ELSIF nMemErr = 1 THEN
	stError.bSTATUS := TRUE;
	stError.nCODE 	:= 4823;
	stError.sSOURCE := 'Incorrect parameter values. Destination address greater that source address';

ELSE
	stError.bSTATUS := TRUE;
	stError.nCODE 	:= 4564;
	stError.sSOURCE := 'Incorrect parameter values. Pointer to destination/source address is NULL or allocated address memory is NULL.';
	END_IF

MemCmpErrExpection := stError.bSTATUS;
END_METHOD

METHOD PROTECTED OutOfBoundsException : BOOL
VAR_INPUT
	nIndex : DINT;
END_VAR
IF (nIndex < 0) OR (nIndex >= THIS^._Count) THEN
	stError.bSTATUS := TRUE;
	stError.nCODE 	:= 5374;
	stError.sSOURCE := 'Out of bounds. You tried to access data outside the range of this list.';
ELSE
	This^.ClearException();
	END_IF
OutOfBoundsException := stError.bSTATUS;
END_METHOD

METHOD TypeMismatchException : BOOL
VAR_INPUT
	Dest,
	Src 	: __SYSTEM.AnyType;
END_VAR
IF Dest.diSize <> Src.diSize THEN
	stError.bSTATUS := TRUE;
	stError.nCODE 	:= 3172;
	stError.sSOURCE := 'Type mismatch. Byte sizes are not the same';
ELSIF Dest.TypeClass <> Src.TypeClass THEN
	stError.bSTATUS := TRUE;
	stError.nCODE 	:= 3172;
	stError.sSOURCE := 'Type mismatch. Type classes are not the same';
ELSE
	THIS^.ClearException();
END_IF
TypeMismatchException := stError.bSTATUS;
END_METHOD

// Copy data from source memory space to desination memory space
METHOD PROTECTED CopyValueTo
VAR_INPUT
	Dest, Src : __SYSTEM.AnyType;
END_VAR
MEMMOVE(Dest.pValue, Src.pValue, TO_UDINT(Dest.diSize));
END_METHOD

// Decrement list size by 1.
METHOD PROTECTED DecrementCount
VAR_INPUT
END_VAR
THIS^.nCount := THIS^.nCount - 1;
END_METHOD

// Deletes/frees node and it's value from memory
METHOD PROTECTED Free_Node
VAR_INPUT
	pNode : POINTER TO ST_NODE; 
END_VAR
__DELETE(pNode^.Data.pValue);
__DELETE(pNode);
END_METHOD

METHOD PROTECTED GetValueAsString : T_MaxString
VAR_INPUT
	 Value : __SYSTEM.AnyType;
END_VAR
VAR	
	pBool			: POINTER TO BOOL;
    pByte			: POINTER TO BYTE;
    pWord			: POINTER TO WORD;
    pDWord			: POINTER TO DWORD;
    pLWord			: POINTER TO LWORD;
    pSint			: POINTER TO SINT;
    pInt			: POINTER TO INT;
    pDint			: POINTER TO DINT;
    pLint			: POINTER TO LINT;
    pUSint			: POINTER TO USINT;
    pUInt			: POINTER TO UINT;
    pUDint			: POINTER TO UDINT;
    pULint			: POINTER TO ULINT;
    pReal			: POINTER TO REAL;
    pLReal			: POINTER TO LREAL;
    pString			: POINTER TO STRING(255);
    pWString		: POINTER TO WSTRING;
    pTime			: POINTER TO TIME;
    pDate			: POINTER TO DATE;
    pDate_And_Time	: POINTER TO DATE_AND_TIME;
    pTime_Of_Day	: POINTER TO TIME_OF_DAY;
    pPointer		: PVOID;
	pLTime 			: POINTER TO LTIME;
END_VAR
IF Value.pValue = 0 THEN GetValueAsString := 'NULL'; RETURN; END_IF;

CASE Value.TypeClass OF 
	__SYSTEM.TYPE_CLASS.TYPE_BOOL:
		pBool := Value.pValue;
		GetValueAsString := TO_STRING(pBool^);
		
    __SYSTEM.TYPE_CLASS.TYPE_BYTE:
		pByte := Value.pValue;
		GetValueAsString := TO_STRING(pByte^);
		
    __SYSTEM.TYPE_CLASS.TYPE_WORD:
		pWord := Value.pValue;
		GetValueAsString := TO_STRING(pWord^);
		
    __SYSTEM.TYPE_CLASS.TYPE_DWORD:
		pDWord := Value.pValue;
		GetValueAsString := TO_STRING(pDWord^);
		
    __SYSTEM.TYPE_CLASS.TYPE_LWORD:
		pLWord := Value.pValue;
		GetValueAsString := TO_STRING(pLWord^);
		
    __SYSTEM.TYPE_CLASS.TYPE_SINT:
		pSint := Value.pValue;
		GetValueAsString := TO_STRING(pSint^);
		
    __SYSTEM.TYPE_CLASS.TYPE_INT:
		pInt := Value.pValue;
		GetValueAsString := TO_STRING(pInt^);
		
    __SYSTEM.TYPE_CLASS.TYPE_DINT:
		pDint := Value.pValue;
		GetValueAsString := TO_STRING(pDint^);
		
    __SYSTEM.TYPE_CLASS.TYPE_LINT:
		pLint := Value.pValue;
		GetValueAsString := TO_STRING(pLint^);
		
    __SYSTEM.TYPE_CLASS.TYPE_USINT:
		pUSint := Value.pValue;
		GetValueAsString := TO_STRING(pUSint^);
		
    __SYSTEM.TYPE_CLASS.TYPE_UINT:
		pUInt := Value.pValue;
		GetValueAsString := TO_STRING(pUInt^);
		
    __SYSTEM.TYPE_CLASS.TYPE_UDINT:
		pUDint := Value.pValue;
		GetValueAsString := TO_STRING(pUDint^);
		
    __SYSTEM.TYPE_CLASS.TYPE_ULINT:
		pULint := Value.pValue;
		GetValueAsString := TO_STRING(pULint^);
		
   __SYSTEM.TYPE_CLASS.TYPE_REAL:
		pReal := Value.pValue;
		GetValueAsString := TO_STRING(pReal^);
		
    __SYSTEM.TYPE_CLASS.TYPE_LREAL:
		pLReal := Value.pValue;
		GetValueAsString := TO_STRING(pLReal^);
		
    __SYSTEM.TYPE_CLASS.TYPE_STRING:
		pString := Value.pValue;
		GetValueAsString := TO_STRING(pString^);
		
   __SYSTEM.TYPE_CLASS.TYPE_WSTRING:
		pWString := Value.pValue;
		GetValueAsString := TO_STRING(pWString^);
		
    __SYSTEM.TYPE_CLASS.TYPE_TIME:
		pTime := Value.pValue;
		GetValueAsString := TO_STRING(pTime^);
		
    __SYSTEM.TYPE_CLASS.TYPE_DATE:
		pDate := Value.pValue;
		GetValueAsString := TO_STRING(pDate^);
		
    __SYSTEM.TYPE_CLASS.TYPE_DATEANDTIME:
		pDate_And_Time := Value.pValue;
		GetValueAsString := TO_STRING(pDate_And_Time^);
		
    __SYSTEM.TYPE_CLASS.TYPE_TIMEOFDAY:
		pTime_Of_Day := Value.pValue;
		GetValueAsString := TO_STRING(pTime_Of_Day^);
	
	__SYSTEM.TYPE_CLASS.TYPE_POINTER:
		GetValueAsString := TO_STRING(Value.pValue);
		
	__SYSTEM.TYPE_CLASS.TYPE_LTIME:
		pLTime := Value.pValue;
		GetValueAsString := TO_STRING(pLTime^);
ELSE
	GetValueAsString := 'TYPE TO STRING CONVERSION NOT SUPPORTED BY THIS TYPE'; 
END_CASE
END_METHOD

// Increments list size by 1
METHOD PROTECTED IncrementCount
VAR_INPUT
END_VAR
THIS^.nCount := THIS^.nCount + 1;
END_METHOD

// Returns pointer to node at specificied location;
METHOD PROTECTED Iterate : POINTER TO ST_NODE
VAR_INPUT
	nIndex : DINT;
END_VAR
VAR 
	i 		: DINT;
	pTemp 	: POINTER TO ST_NODE;
END_VAR
IF THIS^.OutOfBoundsException(nIndex) THEN RETURN; END_IF
IF nIndex = 0 THEN Iterate := THIS^.pHead; RETURN; END_IF
//IF nIndex = THIS^._Count-1 THEN Iterate := pTail; RETURN; END_IF
pTemp := pHead;
FOR i := 1 TO nIndex DO pTemp := pTemp^.pNext; END_FOR
Iterate := pTemp;
END_METHOD

// Allocate memory space for node and the value for it's data on the heap, returns pointer to node;
// WARNING!!! Always have a place to store the node pointer otherwise a memory leak will occur.
METHOD PROTECTED Malloc_Node : POINTER TO ST_NODE
VAR_INPUT
	Variable : __SYSTEM.AnyType;
END_VAR
VAR
	pTemp 	: POINTER TO ST_NODE;
END_VAR
pTemp 					:= __NEW(ST_NODE); // Allocate space in memory for a node.
pTemp^.Data.sValue 		:= THIS^.GetValueAsString(Variable);
pTemp^.Data.pValue 		:= __NEW(BYTE, TO_UDINT(Variable.diSize)); // Allocate space in memory to store data value.
pTemp^.Data.diSize 		:= Variable.diSize;
pTemp^.Data.TypeClass 	:= Variable.TypeClass;

Malloc_Node := pTemp;
END_METHOD

(* Set value of __SYSTEM.Anytype variable *)
METHOD PROTECTED SetValue
VAR_INPUT
	Variable	: __SYSTEM.Anytype;
	Value 		: USINT; // Character/byte to set.
END_VAR
MEMSET(Variable.pValue, Value, TO_UDINT(Variable.diSize));
END_METHOD

(* Checks of list is empty.*)
PROPERTY _Is_Empty : BOOL
GET
_Is_Empty := (THIS^._Count = 0) AND (THIS^.pHead = 0);
END_GET
END_PROPERTY

// Adds an item to the end of the list
METHOD Add_Back : I_List
VAR_INPUT
	Item 	: ANY; // Value to store in list
END_VAR
VAR
	pTemp 	: POINTER TO ST_NODE;
END_VAR
Add_Back := THIS^;
pTemp := THIS^.Malloc_Node(Item);
THIS^.CopyValueTo(pTemp^.Data, Item);

IF THIS^._Is_Empty THEN THIS^.pHead := pTemp;
ELSE Iterate(THIS^._Count - 1)^.pNext := pTemp; END_IF

THIS^.IncrementCount();
END_METHOD

// Adds an item at the front of the list
METHOD Add_Front : I_List
VAR_INPUT
	Item 	: ANY; // Item to store in list
END_VAR
VAR
	pTemp 	: POINTER TO ST_NODE;
END_VAR
Add_Front := THIS^;
pTemp := THIS^.Malloc_Node(Item);
THIS^.CopyValueTo(pTemp^.Data, Item);

pTemp^.pNext := THIS^.pHead; THIS^.pHead := pTemp;
THIS^.IncrementCount();
END_METHOD

(* Empties/Clears/Deletes every item in the list *)
METHOD Clear
VAR
	pTemp : POINTER TO ST_NODE;
END_VAR
pTemp := THIS^.pHead;
WHILE pTemp <> 0 DO
	pTemp := pTemp^.pNext; THIS^.Remove();
END_WHILE
END_METHOD

METHOD FB_exit : BOOL
VAR_INPUT
	(* if TRUE, the exit method is called for exiting an instance that is copied afterwards (online change).*)
	bInCopyCode	: BOOL;
END_VAR
This^.Clear();
END_METHOD

METHOD FB_init : BOOL
VAR_INPUT
	bInitRetains : BOOL; // if TRUE, the retain variables are initialized (warm start / cold start)
	bInCopyCode : BOOL;  // if TRUE, the instance afterwards gets moved into the copy code (online change)
END_VAR
THIS^.Clear();
THIS^.pHead := Tc3_Module.GVL.NULL;
END_METHOD

// Find the location of an item in list.
METHOD Find : I_List
VAR_INPUT
	Item 	: ANY; // Item to find in list
END_VAR
VAR_OUTPUT
	nIndex	: DINT; //Location of item in list 
END_VAR
VAR
	pTemp 	: POINTER TO ST_NODE;
	i 		: DINT;
	n 		: DINT := -1;
END_VAR
Find := THIS^;
IF THIS^.EmptyListException() THEN nIndex := -1; RETURN; END_IF
pTemp := THIS^.pHead;
FOR i := 0 TO THIS^._Count-1 DO
	IF pTemp = 0 THEN EXIT; END_IF
	IF (pTemp^.Data.pValue = 0) 					THEN pTemp := pTemp^.pNext; CONTINUE; END_IF
	IF (Item.TypeClass <> pTemp^.Data.TypeClass) 	THEN pTemp := pTemp^.pNext; CONTINUE; END_IF
	IF (Item.pValue^ <> pTemp^.Data.pValue^) 		THEN pTemp := pTemp^.pNext; CONTINUE; END_IF
	
	CASE Item.TypeClass OF
		__SYSTEM.TYPE_CLASS.TYPE_STRING:
			IF LEN2(Item.pValue) <> LEN2(pTemp^.Data.pValue) THEN pTemp := pTemp^.pNext; CONTINUE; END_IF
			n := MEMCMP(Item.pValue, pTemp^.Data.pValue, LEN2(pTemp^.Data.pValue)+1);
				
		__SYSTEM.TYPE_CLASS.TYPE_WSTRING:
			IF WLEN2(Item.pValue) <> WLEN2(pTemp^.Data.pValue) THEN pTemp := pTemp^.pNext; CONTINUE; END_IF
			n := MEMCMP(Item.pValue, pTemp^.Data.pValue, (WLEN2(pTemp^.Data.pValue)*SIZEOF(WORD))+1);
	ELSE
		IF (Item.diSize <> pTemp^.Data.diSize) THEN pTemp := pTemp^.pNext; CONTINUE; END_IF	
		n := MEMCMP(Item.pValue, pTemp^.Data.pValue, TO_UDINT(Item.diSize));
	END_CASE
	IF n = 0 THEN nIndex := i; RETURN; END_IF
	pTemp := pTemp^.pNext;
	END_FOR
nIndex := -1;
END_METHOD

// Gets item from list at specified location without removing it
METHOD Get : I_List
VAR_INPUT
	Return_Item 	: ANY;  // Variable to store returned item
	nIndex 			: DINT; // Location of item
END_VAR
VAR
	pTemp : POINTER TO ST_NODE;
END_VAR
Get := THIS^;
IF THIS^.EmptyListException() OR THIS^.OutOfBoundsException(nIndex) THEN THIS^.SetValue(Return_Item, 16#0); RETURN; END_IF
pTemp := Iterate(nIndex);
IF THIS^.TypeMismatchException(Return_Item, pTemp^.Data) THEN THIS^.SetValue(Return_Item, 16#0); RETURN; END_IF
THIS^.CopyValueTo(Return_Item, pTemp^.Data);
END_METHOD

// Gets item at the front of the list 
METHOD Get_First : I_List
VAR_INPUT
	Return_Item 	: ANY; // Variable to store returned item
END_VAR
VAR
	pTemp 	: POINTER TO ST_NODE;
END_VAR
Get_First := THIS^;
IF THIS^.TypeMismatchException(Return_Item, pHead^.Data) OR THIS^.EmptyListException() THEN THIS^.SetValue(Return_Item, 16#0); RETURN; END_IF
THIS^.CopyValueTo(Return_Item, pHead^.Data);
Get_First := THIS^;
END_METHOD

// Returns item as a string, if type to string conversion is supported
METHOD Get_Value_As_String : I_List
VAR_INPUT
	nIndex	: DINT; // Location of item
END_VAR
VAR_OUTPUT
	sItem 	: T_MaxString; // Variable to store returned item
END_VAR
VAR
	pTemp : POINTER TO ST_NODE;
END_VAR
Get_Value_As_String := THIS^;
IF THIS^.EmptyListException() OR THIS^.OutOfBoundsException(nIndex) THEN sItem := 'ERR: List is Empty or index Out of Bounds'; RETURN; END_IF
pTemp := Iterate(nIndex);
sItem := pTemp^.Data.sValue;
END_METHOD

// Adds new item to list at specified location, if index = 0, item will be added at the front, if index = count, item will be added at the back
METHOD Insert : I_List
VAR_INPUT
	Item 	: ANY;  // Item to store in list
	nIndex 	: DINT; // Location of item
END_VAR

VAR
	pPrevious 	: POINTER TO ST_NODE;
	pCurrent 	: POINTER TO ST_NODE;
	pTemp 		: POINTER TO ST_NODE;
END_VAR
Insert := THIS^;
IF nIndex = 0 THEN THIS^.Add_Front(Item); RETURN; END_IF
IF nIndex = THIS^._Count THEN THIS^.Add_Back(Item); RETURN; END_IF
IF THIS^.OutOfBoundsException(nIndex) THEN RETURN; END_IF

pTemp := THIS^.Malloc_Node(Item);
THIS^.CopyValueTo(pTemp^.Data, Item);

pPrevious := THIS^.Iterate(nIndex-1);
pCurrent := pPrevious^.pNext;
pPrevious^.pNext := pTemp;
pTemp^.pNext := pCurrent;

THIS^.IncrementCount();
END_METHOD

// Removes item at the front of the list and returns nothing
METHOD Remove : I_List
VAR
	pTemp 	: POINTER TO ST_NODE;
END_VAR
Remove := THIS^;
IF THIS^._Is_Empty THEN RETURN; END_IF

pTemp := THIS^.pHead^.pNext;
THIS^.Free_Node(pHead);
THIS^.pHead := pTemp;

THIS^.DecrementCount();
END_METHOD

// Remove item at specified location and return nothing
METHOD RemoveAt : I_List
VAR_INPUT
	nIndex : DINT; // Location of item
END_VAR
VAR
	pTemp : ARRAY[1..2] OF POINTER TO ST_NODE;
END_VAR
RemoveAt := THIS^;
IF THIS^.EmptyListException() OR THIS^.OutOfBoundsException(nIndex)  THEN RETURN; END_IF
IF nIndex = 0 THEN THIS^.Remove(); RETURN; END_IF

pTemp[1] := THIS^.Iterate(nIndex-1);
pTemp[2] := pTemp[1]^.pNext^.pNext;
THIS^.Free_Node(pTemp[1]^.pNext);
pTemp[1]^.pNext := pTemp[2];

THIS^.DecrementCount();
END_METHOD

// Manually resize list. If list becomes smaller, items on higher locations will be deleted.
METHOD Resize : I_List
VAR_INPUT
	nSize : DINT; // New size of list.
END_VAR
VAR 
	Data 		: __SYSTEM.AnyType;
	nCount,i	: DINT;
END_VAR
Resize := THIS^;
IF nSize <= 0 THEN THIS^.Clear(); RETURN; END_IF
IF nSize = THIS^._Count THEN RETURN; END_IF
IF nSize < THIS^._Count THEN
	nCount := THIS^._Count;
	FOR i := 0 TO nCount - 1 DO
		THIS^.RemoveAt(nCount - 1 - i);
		IF THIS^._Count = nSize THEN RETURN; END_IF
		END_FOR
	END_IF
	
IF nSize > THIS^._Count THEN
	nCount := THIS^._Count;
	FOR i := nCount TO nSize - 1 DO
		THIS^.Add_Back(Data);
		END_FOR
	END_IF
END_METHOD

// Reverses the order of items in the list
METHOD Reverse : I_List
VAR
	pPrevious 	: POINTER TO ST_NODE;
	pCurrent 	: POINTER TO ST_NODE;
	pNext	 	: POINTER TO ST_NODE;
END_VAR
Reverse := THIS^;
pCurrent := pHead;
WHILE pCurrent <> 0 DO
	pNext := pCurrent^.pNext;
	pCurrent^.pNext := pPrevious;
	pPrevious := pCurrent;
	pCurrent := pNext;
END_WHILE
THIS^.pHead := pPrevious;
END_METHOD

// Adds new item to list in the specified location without resizing list
METHOD Set : I_List
VAR_INPUT
	Item 	: ANY; 	// Item to store in list
	nIndex 	: DINT; // Location of item
END_VAR
VAR
	pTemp : POINTER TO ST_NODE;
END_VAR
Set := THIS^;
IF THIS^.OutOfBoundsException(nIndex) THEN RETURN; END_IF
pTemp := Iterate(nIndex);
IF THIS^.TypeMismatchException(pTemp^.Data, Item) THEN RETURN; END_IF
THIS^.CopyValueTo(pTemp^.Data, Item);
END_METHOD

END_FUNCTION_BLOCK

// POUs/Examples/P_Queue_Example
// Login into PLC and live write eState. Try nData and nRTNData once your done. eState Initialises at IDLE
PROGRAM P_Queue_Example
VAR
	fbList 		: FB_LIST;
	fbQueue 	: FB_Queue;
	sData 		: STRING;
	sRTNData	: ARRAY[0..3] OF STRING; //returned data
	nData 		: DINT;
	nRTNData 	: ARRAY[0..3] OF DINT; 
	nCount 		: DINT;
	eState 		: (IDLE, ENQUEUE_AND_PEEK, GET_ITEM_COUNT,REVERSE_AND_PEEK, DEQUEUE_AND_PEEK, CLEAR_Q);
	stError 	: ST_ERROR;
END_VAR

fbQueue(ipList := fbList);
stError := fbQueue._Error_Status;
CASE eState OF
	ENQUEUE_AND_PEEK: //
		sData := 'Cats';fbQueue.Enqueue(sData);
		sData := 'Dogs';fbQueue.Enqueue(sData);
		sData := 'Birds';fbQueue.Enqueue(sData);
		sData := 'Fish';fbQueue.Enqueue_At_Front(sData);

		fbQueue.Peek(sRTNData[0], 0)
			   .Peek(sRTNData[1], 1)
			   .Peek(sRTNData[2], 2)
			   .Peek(sRTNData[3], 3);
		eState := IDLE;
		
	GET_ITEM_COUNT: 
		nCount := fbQueue._Count;
		eState := IDLE;
		
	REVERSE_AND_PEEK:
		fbQueue.Reverse()
			   .Peek(sRTNData[0], 0)
			   .Peek(sRTNData[1], 1)
			   .Peek(sRTNData[2], 2)
			   .Peek(sRTNData[3], 3);
		eState := IDLE;
	
	DEQUEUE_AND_PEEK:
		fbQueue.Dequeue(sRTNData[0])
			   .Dequeue_Void()
			   .Peek(sRTNData[1], 1)
			   .Peek(sRTNData[2], 2)
			   .Peek(sRTNData[3], 3);
		eState := IDLE;
		
	CLEAR_Q:
		fbQueue.Clear();
		eState := IDLE;	
END_CASE

END_PROGRAM

// POUs/Function Blocks/FB_Queue
FUNCTION_BLOCK FB_Queue EXTENDS FB_Collections  IMPLEMENTS I_Queue
VAR_INPUT
	ipList : I_List; // List to perform operations on.
END_VAR
VAR
	//ipItems_List : I_List; // List holding items on the queue
END_VAR

(* Number of items in queue*)
PROPERTY _Count : DINT
GET
_Count := THIS^.ipList._Count;
END_GET
END_PROPERTY

(* Checks of queue is empty.*)
PROPERTY _Is_Empty : BOOL
GET
_Is_Empty := THIS^.ipList._Is_Empty;
END_GET
END_PROPERTY

METHOD PROTECTED CatchError : BOOL
VAR_INPUT
END_VAR
//THIS^.ipItems_List(stError => THIS^.stError);
THIS^.stError := ipList._Error_Status;
CatchError := stError.bSTATUS;
END_METHOD

(* Empties/Clears/Deletes every item on the queue*)
METHOD Clear
THIS^.ipList.Clear();
END_METHOD

(* Gets and remove item at the front of the queue *)
METHOD Dequeue : I_Queue
VAR_INPUT
	Item : ANY; (* Variable to store returned item value *)
END_VAR
Dequeue := THIS^;
THIS^.ipList.Get_First(Item);
IF THIS^.CatchError() THEN RETURN; END_IF;
THIS^.ipList.Remove();
THIS^.CatchError();
END_METHOD

(* Removes item at the front of the queue without returning anything *)
METHOD Dequeue_Void : I_Queue
VAR_INPUT
END_VAR
Dequeue_Void := THIS^;
THIS^.ipList.Remove();
THIS^.CatchError();
END_METHOD

(* Adds item at the back of the queue *)
METHOD Enqueue : I_Queue
VAR_INPUT
	Item : ANY; (* Variable containg data to store on the queue *)
END_VAR
Enqueue := THIS^;
THIS^.ipList.Add_Back(Item);
THIS^.CatchError();
END_METHOD

(* Adds item at the front of the queue *)
METHOD Enqueue_At_Front : I_Queue
VAR_INPUT
	Item : ANY; (* Variable containg data to store on the queue *)
END_VAR
Enqueue_At_Front := THIS^;
THIS^.ipList.Add_Front(Item);
THIS^.CatchError();
END_METHOD

(* Get item from the queue without removing it. *)
METHOD Peek : I_Queue
VAR_INPUT
	Item 	: ANY; (* Variable to store returned item value *)
	nIndex 	: DINT; (* Location of item*)
END_VAR
Peek := THIS^;
THIS^.ipList.Get(Item, nIndex);
THIS^.CatchError();
END_METHOD

METHOD Reverse : I_Queue
VAR_INPUT
END_VAR
Reverse := THIS^;
THIS^.ipList.Reverse();
THIS^.CatchError();
END_METHOD

END_FUNCTION_BLOCK

// POUs/Examples/P_Stack_Example
// Login into PLC and live write eState. Try nData and nRTNData once your done. eState Initialises at IDLE
PROGRAM P_Stack_Example
VAR
	fbList 		: FB_LIST;
	fbStack 	: FB_Stack;
	sData 		: STRING;
	sRTNData	: ARRAY[0..3] OF STRING; //returned data
	nData 		: DINT;
	nRTNData 	: ARRAY[0..3] OF DINT; 
	nCount 		: DINT;
	eState 		: (IDLE, PUSH_AND_PEEK, GET_ITEM_COUNT,REVERSE_AND_PEEK, POP, CLEAR_STACK);
	stError 	: ST_ERROR;
END_VAR

fbStack(ipList := fbList);
stError := fbStack._Error_Status;
CASE eState OF
	PUSH_AND_PEEK:
		sData := 'Cats';fbStack.Push(sData);
		sData := 'Dogs';fbStack.Push(sData);
		sData := 'Birds';fbStack.Push(sData);
		sData := 'Fish';fbStack.Push(sData);

		fbStack.Peek(sRTNData[0], 0)
			   .Peek(sRTNData[1], 1)
			   .Peek(sRTNData[2], 2)
			   .Peek(sRTNData[3], 3);
		eState := IDLE;
		
	GET_ITEM_COUNT: 
		nCount := fbStack._Count;
		eState := IDLE;
		
	REVERSE_AND_PEEK:
		fbStack.Reverse()
			   .Peek(sRTNData[0], 0)
			   .Peek(sRTNData[1], 1)
			   .Peek(sRTNData[2], 2)
			   .Peek(sRTNData[3], 3);
		eState := IDLE;
	
	POP:
		fbStack.Pop(sRTNData[0])
			   .Pop(sRTNData[1])
			   .Pop(sRTNData[2]);
		eState := IDLE;
		
	CLEAR_STACK:
		fbStack.Clear();
		eState := IDLE;	
END_CASE

END_PROGRAM

// POUs/Function Blocks/FB_Stack
FUNCTION_BLOCK FB_Stack EXTENDS FB_Collections IMPLEMENTS I_Stack
VAR_INPUT
	ipList : I_List; // List to perform operations on.
END_VAR
VAR_OUTPUT
END_VAR

(* Number of elements in the stack *)
PROPERTY _Count : DINT
GET
_Count := THIS^.ipList._Count;
END_GET
END_PROPERTY

(* Checks of stack is empty.*)
PROPERTY _Is_Empty : BOOL
GET
_Is_Empty := THIS^.ipList._Is_Empty;
END_GET
END_PROPERTY

METHOD PROTECTED CatchError : BOOL
VAR_INPUT
END_VAR
stError := THIS^.ipList._Error_Status;
CatchError := stError.bSTATUS;
END_METHOD

(* Empties/Clears/Deletes every item on the stack*)
METHOD Clear
VAR_INPUT
END_VAR
THIS^.ipList.Clear();
END_METHOD

(* Get item from stack without removing it. *)
METHOD Peek : I_Stack
VAR_INPUT
	Item 	: ANY; (* Variable to store returned item value *)
	nIndex 	: DINT; (* Location of item*)
END_VAR
Peek := THIS^;
THIS^.ipList.Get(Item, nIndex);
THIS^.CatchError();
END_METHOD

(* Gets and deletes item at the top of the stack *)
METHOD Pop : I_Stack
VAR_INPUT
	Item : ANY; (* Variable to store returned item value *)
END_VAR
Pop := THIS^;
THIS^.ipList.Get_First(Item);
IF THIS^.CatchError() THEN RETURN; END_IF;
THIS^.ipList.Remove();
THIS^.CatchError();
END_METHOD

(* Removes item at the top of the stack without returning anything *)
METHOD Pop_Void : I_Stack
VAR_INPUT
END_VAR
Pop_Void := THIS^;
THIS^.ipList.Remove();
THIS^.CatchError();
END_METHOD

(* Add item to the top of the stack *)
METHOD Push : I_Stack
VAR_INPUT
	Item : ANY; (* Variable containg data to store on the stack *)
END_VAR
Push := THIS^;
THIS^.ipList.Add_Front(Item);
THIS^.CatchError();
END_METHOD

(* Reverses order of items on stack *)
METHOD Reverse : I_Stack
VAR_INPUT
END_VAR
Reverse := THIS^;
THIS^.ipList.Reverse();
THIS^.CatchError();
END_METHOD

(* Get item at the top of the stack without removing it. *)
METHOD Top : I_Stack
VAR_INPUT
	Item 	: ANY; (* Variable to store returned item value *)
END_VAR
Top := THIS^;
THIS^.ipList.Get_First(Item);
IF THIS^.CatchError() THEN RETURN; END_IF;
END_METHOD

END_FUNCTION_BLOCK

// POUs/MAIN
PROGRAM MAIN
VAR
END_VAR

P_Array_List_Example();
P_List_Example();
P_Queue_Example();
P_Stack_Example();

END_PROGRAM

// Project Information/F_GetCompany
// This function has been automatically generated from the project information.
{attribute 'signature_flag' := '1073741824'}
{attribute 'TcGenerated'}
{attribute 'no-analysis'}
FUNCTION F_GetCompany : WSTRING
VAR_INPUT
	
END_VAR

F_GetCompany := "FisoThemes";

END_FUNCTION

// Project Information/F_GetTitle
// This function has been automatically generated from the project information.
{attribute 'signature_flag' := '1073741824'}
{attribute 'TcGenerated'}
{attribute 'no-analysis'}
FUNCTION F_GetTitle : WSTRING
VAR_INPUT
	
END_VAR

F_GetTitle := "TwinCat Dynamic Collections";

END_FUNCTION

// Project Information/F_GetVersion
// This function has been automatically generated from the project information.
{attribute 'signature_flag' := '1073741824'}
{attribute 'TcGenerated'}
{attribute 'no-analysis'}
FUNCTION F_GetVersion : ST_LibVersion
VAR_INPUT
	
END_VAR

F_GetVersion.iMajor := 0;
F_GetVersion.iMinor := 2;
F_GetVersion.iBuild := 0;
F_GetVersion.iRevision := 0;

END_FUNCTION
